Universal Robots PolyScope program: Cobot_soudure_28112023.urp

Program Cobot_soudure_28112023 (installation=Cobot_soudure_28112023 directory=/home/ur/ursim/ursim-5.11.0.108249/programs/TRAVAIL 27112023 createdIn=5.9.4.1031232 lastSavedIn=5.11.0.108249 robotSerialNumber=20195299999)
Calibrated DH parameters: a=[0, -0.6127, -0.57155, 0, 0, 0]; d=[0.1807, 0, 0, 0.17415, 0.11985, 0.11655]; alpha=[1.570796, 0, 0, 1.570796, -1.570796, 0]; deltaTheta=[0, 0, 0, 0, 0, 0]
InitVariablesNode variables(variable(name=Test_Gaz, expression=False), variable(name=Test_Job, expression=False), variable(name=Test_Ordre_Mar, expression=False), variable(name=Valide_Gaz, expression=False), variable(name=fin_soud, expression=1), variable(name=secu_d, expression=0), variable(name=secu_g, expression=0), variable(name=timer_ret_gaz, expression=0))
BeforeStart
  Folder fonctions
    Folder Init [hidden by the author, left out]
    Folder Diverses [hidden by the author, left out]
    Folder Demande [hidden by the author, left out]
    Folder Configuration [hidden by the author, left out]
    Folder Execution [hidden by the author, left out]
    Folder Pas_A_Pas [hidden by the author, left out]
    Folder PopUps [hidden by the author, left out]
    Folder Mouvements soudures [hidden by the author, left out]
    Folder General [hidden by the author, left out]
Robot Program (runOnlyOnce=true)
  SuppressedNode
    Script file /home/ur/ursim/ursim-5.11.0.108249/programs/SCRIPT/Scripts_soudure/general.script
      | while (True):
      |   # 68 "Programme de robot"
      |   global safe_mode=0
      | 
      |   set_configurable_digital_out(0, False)
      |   set_configurable_digital_out(1, False)
      | 
      |   while (get_configurable_digital_in(4) ==   True    or  get_configurable_digital_in(5) ==   True  ):
      | 
      |     sync()
      |     # 94 "'clingottement pour signifier qu'il y  un defaut sur un des carters '"
      |     set_standard_digital_out(4, False)
      |     set_configurable_digital_out(6, False)
      |     sleep(0.5)
      |     set_standard_digital_out(4, True)
      |     set_configurable_digital_out(6, True)
      |     sleep(0.5)
      |     sync()
      |   end
      | 
      |   set_configurable_digital_out(6, False)
      |   set_standard_digital_out(4, False)
      |   sleep(2.0)
      |   #movel(pose_add(get_target_tcp_pose(), pose_sub(PointPassage_12_to_p, PointPassage_12_from_p)), a=0.01, v=2.0E-4)
      |   global angle_base= get_actual_joint_positions ()
      |   if (angle_base[0]  <= 0.7):
      |     if (angle_base[0] >= 1.6):
      |       # 116 "Départ"        A CHANGER PAR UNE POSTION ENREGISTREE
      |       movej(pose_depart, a=accelerationHorsSoudure, v=vitesseHorsSoudure)
      |     else:
      |       if (angle_base[0]>1.6):
      |         movej(Point_init_D, a=accelerationHorsSoudure, v=vitesseHorsSoudure)
      |         movej(Point_avt_initD, a=accelerationHorsSoudure, v=vitesseHorsSoudure)
      |       else:
      |         if (angle_base[0]<0.7):
      |           movej(Point_init_G, a=accelerationHorsSoudure, v=vitesseHorsSoudure)
      |         end
      |       end
      |     end
      |   else:
      |     # 124 "SinonSi angle_base[0]>1.6"
      |     if (angle_base[0]>1.6):
      | 
      |       movej(Point_init_D, a=accelerationHorsSoudure, v=vitesseHorsSoudure)
      |       movej(Point_avt_initD, a=accelerationHorsSoudure, v=vitesseHorsSoudure)
      |     else:
      |       if (angle_base[0]<0.7):
      |         movej(Point_init_G, a=accelerationHorsSoudure, v=vitesseHorsSoudure)
      |       end
      |     end
      |   end
      |   # 131 "Départ"             A CHANGER PAR UNE POSTION ENREGISTREE
      |   movej(pose_depart, a=accelerationHorsSoudure, v=vitesseHorsSoudure)
      |   global angle_base= get_actual_joint_positions ()
      |   # 'mode config'
      |   if (get_configurable_digital_in(7)  ==   False    and  get_standard_digital_in(7)  ==   False  ):
      |     if ((config_g  ==  1)   and   (config_d  ==  1)):
      |       pop_up_config_g_et_d()
      |     else:
      |       if ((config_g  == 1)):
      |         pop_up_config_g()
      |       else:
      |         if (config_d  ==  1):
      |           pop_up_config_d()
      |         else:
      |           if ((config_g  ==  0)  and  (config_d  ==  0)):
      |             pop_up_config()
      |           end
      |         end
      |       end
      |     end
      |     global boucle=1
      |     while ((get_configurable_digital_in(7)  ==   False  )  and  (boucle  ==  1)   and  (get_standard_digital_in(7) ==   False  )):
      |       thread Thread_while_145():
      |         while (True):
      |           set_standard_digital_out(5, True)
      |           set_standard_digital_out(6, False)
      |           sleep(0.5)
      |           set_standard_digital_out(5, False)
      |           set_standard_digital_out(6, True)
      |           sleep(0.5)
      |           sync()
      |         end
      |       end
      |       if (get_standard_digital_in(3) ==   False    and  get_standard_digital_in(2) ==   False    and  get_configurable_digital_in(add_bp_ConfigReglage)  ==    False    and  get_standard_digital_in(add_bp_ConfigReglage) ==   False  ):
      |         global thread_handler_145=run Thread_while_145()
      |         while (get_standard_digital_in(3) ==   False    and  get_standard_digital_in(2) ==   False    and  get_configurable_digital_in(add_bp_ConfigReglage)  ==    False    and  get_standard_digital_in(add_bp_ConfigReglage) ==   False  ):
      |           sync()
      |         end
      |         kill thread_handler_145
      |       end
      |       if (get_standard_digital_in(2)  ==   True  ):
      |         set_standard_digital_out(5, True)
      |         set_standard_digital_out(6, False)
      |         movej(Point_init_G, a=accelerationHorsSoudure, v=vitesseHorsSoudure, r=0.006)
      |         movej(Point_Attente_G, a=accelerationHorsSoudure, v=vitesseHorsSoudure, r=0.006)
      |         movej(Point_config_g, a=accelerationHorsSoudure, v=vitesseHorsSoudure)
      |         global led_cobot=1
      |         fun_config_g()
      |         global led_cobot=0
      |         fun_valid_config_g()
      |         movej(Point_Attente_G, a=accelerationHorsSoudure, v=vitesseHorsSoudure, r=0.006)
      |         movej(Point_init_G, a=accelerationHorsSoudure, v=vitesseHorsSoudure, r=0.006)
      |         # 170 "Départ"         A CHANGER PAR UNE POSTION ENREGISTREE
      |         movej(pose_depart, a=accelerationHorsSoudure, v=vitesseHorsSoudure)
      |       end
      | 
      |       if (get_standard_digital_in(3)  ==   True  ):
      |         set_standard_digital_out(6, True)
      |         set_standard_digital_out(5, False)
      |         movej(Point_avt_initD, a=accelerationHorsSoudure, v=vitesseHorsSoudure, r=0.006)
      |         movej(Point_init_D, a=accelerationHorsSoudure, v=vitesseHorsSoudure)
      |         movej(Point_Attente_D, a=accelerationHorsSoudure, v=vitesseHorsSoudure, r=0.006)
      |         movej(Point_config_d, a=accelerationHorsSoudure, v=vitesseHorsSoudure)
      |         global led_cobot=1
      |         fun_config_d()
      |         global led_cobot=0
      |         fun_valid_config_d()
      |         movej(Point_Attente_D, a=accelerationHorsSoudure, v=vitesseHorsSoudure, r=0.006)
      |         movej(Point_init_D, a=accelerationHorsSoudure, v=vitesseHorsSoudure, r=0.006)
      |         movej(Point_avt_initD, a=accelerationHorsSoudure, v=vitesseHorsSoudure, r=0.006)
      |         # 190 "Départ"         A CHANGER PAR UNE POSTION ENREGISTREE
      |         movej(pose_depart, a=accelerationHorsSoudure, v=vitesseHorsSoudure)
      |       end
      |     end
      |   end
      |   # '"Reglage"'
      | 
      |   if (get_configurable_digital_in(add_bp_ConfigReglage)  ==   False    and  get_standard_digital_in(add_bp_ConfigReglage)  ==   True  ):
      |     if ((config_g  ==  1)   and   (config_d  ==  1)):
      |       pop_up_reg_gd()
      |       global boucle=1
      |     else:
      |       if (config_g  ==  1):
      |         pop_up_reg_gd()
      |         global boucle=1
      |       else:
      |         if (config_d  ==  1):
      |           pop_up_reg_d()
      |           global boucle=1
      |         else:
      |           close_popup()
      |           while (get_standard_digital_in(add_bp_ConfigReglage)  ==   True  ):
      |             popup("Aucune configuration n'est actuellement detectée.", "Erreur", False, True, blocking=True)
      |           end
      |         end
      |       end
      |     end
      |     global boucle=1
      |     while ((get_configurable_digital_in(add_bp_ConfigReglage)  ==   False  )  and  (boucle  ==  1)   and  (get_standard_digital_in(add_bp_ConfigReglage) ==   True  )):
      |       thread Thread_while_208():
      |         while (True):
      |           if (config_g  ==  1):
      |             set_standard_digital_out(5, True)
      |           end
      |           if (config_d  ==  1):
      |             set_standard_digital_out(6, True)
      |           end
      |           sleep(0.5)
      |           set_standard_digital_out(5, False)
      |           set_standard_digital_out(6, False)
      |           sleep(0.5)
      |         end
      |       end
      |       if (get_standard_digital_in(3) ==   False    and  get_standard_digital_in(2) ==   False    and  get_configurable_digital_in(7)  ==    False    and  get_standard_digital_in(7)  ==   True  ):
      |         global thread_handler_208=run Thread_while_208()
      |         while (get_standard_digital_in(3) ==   False    and  get_standard_digital_in(2) ==   False    and  get_configurable_digital_in(7)  ==    False    and  get_standard_digital_in(7)  ==   True  ):
      |           sync()
      |         end
      |         kill thread_handler_208
      |       end
      |       if (get_standard_digital_in(2)  ==   True  ):
      |         global safe_mode=1
      |         set_standard_digital_out(5, True)
      |         set_standard_digital_out(6, False)
      |         movej(Point_init_G, a=accelerationHorsSoudure, v=vitesseHorsSoudure, r=0.006)
      |         movej(Point_Attente_G, a=accelerationHorsSoudure, v=vitesseHorsSoudure, r=0.006)
      |         movej(pose_inter_g, a=accelerationHorsSoudure, v=vitesseHorsSoudure)
      |         global led_cobot=1
      |         fun_Pas_A_Pas_g()
      |         global led_cobot=0
      |         global safe_mode=0
      |         global boucle=0
      |       end
      |       if (get_standard_digital_in(3)  ==   True  ):
      |         global safe_mode=1
      |         set_standard_digital_out(6, True)
      |         set_standard_digital_out(5, False)
      |         movej(Point_avt_initD, a=accelerationHorsSoudure, v=vitesseHorsSoudure, r=0.006)
      |         movej(Point_init_D, a=accelerationHorsSoudure, v=vitesseHorsSoudure, r=0.006)
      |         movej(pose_inter_d, a=accelerationHorsSoudure, v=vitesseHorsSoudure)
      |         global led_cobot=1
      |         fun_Pas_A_Pas_d()
      |         global led_cobot=0
      |         global safe_mode=0
      |         global boucle=0
      |       end
      |     end
      |   end
      |   # 'mode execution'
      |   if (get_configurable_digital_in(add_bp_ConfigReglage)  ==   True  ):
      |     if ((config_g  ==  1)   and   (config_d  ==  1)):
      |       pop_up_exe()
      |       global boucle=1
      |     else:
      |       if (config_g  ==  1):
      |         pop_up_exe_g()
      |         global boucle=1
      |       else:
      |         if (config_d  ==  1):
      |           pop_up_exe_d()
      |           global boucle=1
      |         else:
      |           close_popup()
      |           while (get_configurable_digital_in(add_bp_ConfigReglage)  ==   True  ):
      |             popup("Aucune programmation n'est actuellement detectée, veillez à programmer une pièce avant de vouloir l'éxécuter.", "Erreur", False, True, blocking=True)
      |           end
      |         end
      |       end
      |     end
      |     while (( get_configurable_digital_in(add_bp_ConfigReglage)  ==   True  )   and  (boucle  ==  1)):
      |       thread Thread_while_259():
      |         while (True):
      |           if (config_g  ==  1):
      |             set_standard_digital_out(5, True)
      |           end
      |           if (config_d  ==  1):
      |             set_standard_digital_out(6, True)
      |           end
      |           sleep(0.5)
      |           set_standard_digital_out(5, False)
      |           set_standard_digital_out(6, False)
      |           sleep(0.5)
      |         end
      |       end
      |       if (get_standard_digital_in(3) ==   False    and  get_standard_digital_in(2) ==   False    and  get_configurable_digital_in(add_bp_ConfigReglage) ==   True  ):
      |         global thread_handler_259=run Thread_while_259()
      |         while (get_standard_digital_in(3) ==   False    and  get_standard_digital_in(2) ==   False    and  get_configurable_digital_in(add_bp_ConfigReglage) ==   True  ):
      |           sync()
      |         end
      |         kill thread_handler_259
      |       end
      |       if ((get_standard_digital_in(2)  ==   True  )  and  (config_g  ==   True  )):
      |         global boucle_g=1
      |         while (boucle_g  ==  1):
      |           set_configurable_digital_out(0, True)
      |           set_standard_digital_out(5, True)
      |           set_standard_digital_out(6, False)
      |           sleep(0.25)
      |           set_standard_digital_out(5, False)
      |           sleep(0.25)
      |           if (get_configurable_digital_in(4)  ==    False  ):
      |             set_standard_digital_out(5, True)
      |             if (get_configurable_digital_in(4)  ==    False  ):
      |               close_popup()
      |               while (get_configurable_digital_in(4) == False):
      |                 sync()
      |               end
      |             end
      |           end
      |           if (get_configurable_digital_in(4)  ==    True  ):
      |             global secu_g=1
      |             set_standard_digital_out(5, True)
      |             movej(Point_init_G, a=accelerationHorsSoudure, v=vitesseHorsSoudure, r=0.006)
      |             fun_execution_g()
      |             movej(Point_Attente_G, a=accelerationHorsSoudure, v=vitesseHorsSoudure, r=0.006)
      |             movej(Point_init_G, a=accelerationHorsSoudure, v=vitesseHorsSoudure, r=0.006)
      |             # 294 "Départ"         A CHANGER PAR UNE POSTION ENREGISTREE
      |             movej(pose_depart, a=accelerationHorsSoudure, v=vitesseHorsSoudure)
      |             set_configurable_digital_out(0, False)
      |             global secu_g=0
      |             global boucle_g=0
      |           end
      |         end
      |         global boucle=0
      |       else:
      |         if ((get_standard_digital_in(2)  ==   True  )  and  (config_g  ==   False  )):
      |           close_popup()
      |           popup("Aucune programmation n'est actuellement detectée sur la table gauche, veillez à programmer une pièce avant de vouloir l'éxécuter.", "Erreur", False, True, blocking=True)
      |           global boucle=0
      |         end
      |       end
      |       if ((get_standard_digital_in(3)  ==   True  )  and  (config_d  ==   True  )):
      |         global boucle_d=1
      |         pop_up_deb_exe_d()
      |         while (boucle_d  ==  1):
      |           set_configurable_digital_out(1, True)
      |           set_standard_digital_out(5, False)
      |           set_standard_digital_out(6, True)
      |           sleep(0.25)
      |           set_standard_digital_out(6, False)
      |           sleep(0.25)
      |           if (get_configurable_digital_in(5)  ==    False  ):
      |             set_standard_digital_out(6, True)
      |             sleep(6.0)
      |             if (get_configurable_digital_in(5)  ==    False  ):
      |               close_popup()
      |               while (get_configurable_digital_in(5) == False):
      |                 sync()
      |               end
      |             end
      |           end
      |           if (get_configurable_digital_in(5)  ==    True  ):
      |             global secu_d=1
      |             set_standard_digital_out(6, True)
      |             movej(Point_avt_initD, a=accelerationHorsSoudure, v=vitesseHorsSoudure)
      |             fun_execution_d()
      |             set_configurable_digital_out(1, False)
      |             global secu_d=0
      |             global boucle_d=0
      |           end
      |         end
      |         global boucle=0
      |       else:
      |         if ((get_standard_digital_in(3)  ==   True  )  and  (config_d  ==   False  )):
      |           close_popup()
      |           popup("Aucune programmation n'est actuellement detectée sur la table droite, veillez à programmer une pièce avant de vouloir l'éxécuter.", "Erreur", False, True, blocking=True)
      |           global boucle=0
      |         end
      |       end
      |     end
      |   end
      | end
      | end
  Script: General()
SubProgram Recopie_Table_Droite (keepSynchronizedWithDisk=false)
  SuppressedNode
    URCap Path (Robotiq_Copilot, Robotiq Inc.) dataModel(NodeInitializedKey=true, urcapVersion=1.14.3, pathOptionsTypeKey=TOOL_ON_ROBOT, HackTriggeringContributionIsDefinedMethodKey=true, version=1.14.3.2973, trajectoryPath={}); state(isChildrenLocked=true)
      URCap BeforeStart Node (Robotiq_Copilot, Robotiq Inc.)
        'Insert nodes below.'
  Popup Message (haltProgram=false message=Recopie sur la table de droite  inputType=Text)
SubProgram Recopie_Table_Gauche (keepSynchronizedWithDisk=false)
  SuppressedNode
    URCap Path (Robotiq_Copilot, Robotiq Inc.) dataModel(NodeInitializedKey=true, urcapVersion=1.14.3, pathOptionsTypeKey=TOOL_ON_ROBOT, HackTriggeringContributionIsDefinedMethodKey=true, version=1.14.3.2973, trajectoryPath={}); state(isChildrenLocked=true)
      URCap BeforeStart Node (Robotiq_Copilot, Robotiq Inc.)
        'Insert nodes below.'
  Popup Message (haltProgram=false message=Recopie sur la table de gauche inputType=Text)
Thread Thread_1 (runOnlyOnce=false)
  Folder Test_Ordre_Marche [hidden by the author, left out]
  Script: sync()
Thread Thread_2 (runOnlyOnce=false)
  Folder mode_soudure [hidden by the author, left out]
  Script: sync()
Thread Thread_3 (runOnlyOnce=false)
  Folder led_cobot_2 [hidden by the author, left out]
  Script: sync()
Thread Thread_4 (runOnlyOnce=false)
  Folder led_cobot [hidden by the author, left out]
  Script: sync()
Thread Thread_5 (runOnlyOnce=false)
  Folder Test_Arc_On [hidden by the author, left out]
  Script: sync()
Thread Thread_6 (runOnlyOnce=false)
  Folder Test_Job [hidden by the author, left out]
  Script: sync()
Thread Thread_7 (runOnlyOnce=false)
  Folder secu [hidden by the author, left out]
  Script: sync()
Thread Thread_8 (runOnlyOnce=false)
  Folder bloq_soud_arret [hidden by the author, left out]
  SuppressedNode
    Folder freedrive_droit
      If led_cobot ≟  True
        If tool_in[1] ≟ True
          Script: teach_mode()
        Else 
          Script: end_teach_mode()
  Script: sync()
SuppressedNode
  Thread Thread_9 (runOnlyOnce=false)
    Folder reglage
      If reglage_d ≠0
        Script file /programs/Programmes/cobot_v2/sript/Part_reglage/REGLAGE_D.script
          |     ##############################################################################
          | 
          | ########################soudure point#########################################
          | 
          |     ##############################################################################
          | 
          |         if reglage_d == 1:                                    #remplissage tableau
          |             teach_mode()
          |             fun_popup_soud(1, 1, i)
          |             fun_front_up(adresse_bp_cobot)
          |             tab_point_app_d[i] =  get_actual_tcp_pose()     #Enregistrer position dans tableau d'approche des soudue points quand appui bouton
          |             close_popup()
          | 
          |             fun_popup_soud(2, 1, i)
          |             fun_front_up(adresse_bp_cobot)
          |             tab_point_deb_d[i] =  get_actual_tcp_pose()     #Enregistrer position debut quand appui bouton bp_cobot
          |             close_popup()
          | 
          |             tab_point_ret_d[i] = tab_point_app_d[i]         #point de retrait est le meme que le point d approche
          |             end_teach_mode()
          |             global reconfig = 1
          |             global reglage_d = 0
          | 
          |             sync()
          | 
          |         ##############################################################################
          | 
          |     ##############################################################################
          | 
          | ########################soudure lineaire######################################
          | 
          |     ##############################################################################
          | 
          |         elif reglage_d == 2:                		            #remplissage tableau
          |             teach_mode()
          |             fun_popup_soud(1, 2, j)
          |             fun_front_up(adresse_bp_cobot)
          |             tab_lin_app_d[j] =  get_actual_tcp_pose()     	#Enregistrer position dans tableau d approche des soudures lineaire quand appui Bp_cobot
          |             close_popup()
          | 
          |             fun_popup_soud(2, 2, j)
          |             fun_front_up(adresse_bp_cobot)
          |             tab_lin_deb_d[j] =  get_actual_tcp_pose()     	#Enregistrer position dans tableau debut quand appui Bp_cobot
          |             close_popup()
          | 
          |             fun_popup_soud(6, 2, j)
          |             fun_front_up(adresse_bp_cobot)
          |             tab_lin_fin_d[j] =  get_actual_tcp_pose()     	#Enregistrer position dans un tableau fin quand appui Bp_cobot
          |             close_popup()
          | 
          |             vit_lin_d[j] = fun_demande_vit(2)
          | 
          |             fun_popup_soud(7, 2, j)
          |             fun_front_up(adresse_bp_cobot)
          |             tab_lin_ret_d[j] =  get_actual_tcp_pose()     	#Enregistrer position dans tableau retrait quand appui Bp_cobot
          |             close_popup()
          |             end_teach_mode()
          |             global reglage_d = 0
          | 
          |             sync()
          | 
          |         ##############################################################################
          | 
          |     ##############################################################################
          | 
          | #########################soudure arc de cercle##################################
          | 
          |     #################################################################################
          | 
          |         elif reglage_d == 3:                                  #remplissage tableau
          |             teach_mode()
          |             fun_popup_soud(1, 3, k)
          |             fun_front_up(adresse_bp_cobot)
          |             tab_arc_app_d[k] =  get_actual_tcp_pose() 	    #Enregistrer position dans tableau d approche des soudures arc de cercle quand appui
          |             close_popup()
          | 
          |             fun_popup_soud(2, 3, k)
          |             fun_front_up(adresse_bp_cobot)
          |             tab_arc_deb_d[k] =  get_actual_tcp_pose() 	    #Enregistrer position dans tableau debut quand appui Bp_d
          |             close_popup()
          | 
          |             fun_popup_soud(4, 3, k)
          |             fun_front_up(adresse_bp_cobot)
          |             tab_arc_mil_d[k] =  get_actual_tcp_pose() 	    #Enregistrer position dans tableau milieu quand appui Bp_cobot
          |             close_popup()
          | 
          |             fun_popup_soud(6, 3, k)
          |             fun_front_up(adresse_bp_cobot)
          |             tab_arc_fin_d[k] =  get_actual_tcp_pose() 	    #Enregistrer position dans un tableau fin quand appui Bp_cobot
          |             close_popup()
          | 
          |             vit_arc_d[k] = fun_demande_vit(3)               #demande de vitesse des soudures lineaire
          | 
          |             fun_popup_soud(7, 3, k)
          |             fun_front_up(adresse_bp_cobot)
          |             tab_arc_ret_d[k] =  get_actual_tcp_pose() 	    #Enregistrer position dans tableau retrait quand appui Bp_cobot
          |             close_popup()
          |             end_teach_mode()
          |             global reglage_d = 0
          | 
          |             sync()
          | 
          |         ##############################################################################
          | 
          |     ##############################################################################
          | 
          | ############################soudure cercle####################################
          | 
          |     #################################################################################
          | 
          |         elif reglage_d == 4:                                  #remplissage tableau
          |             teach_mode()
          |             fun_popup_soud(1, 4, l)
          |             fun_front_up(adresse_bp_cobot)
          |             tab_cer_app_d[l] =  get_actual_tcp_pose()     	#Enregistrer position dans tableau d approche des soudures arc de cercle quand appui Bp_cobot
          |             close_popup()
          | 
          |             fun_popup_soud(2, 4, l)
          |             fun_front_up(adresse_bp_cobot)
          |             tab_cer_deb_d[l] =  get_actual_tcp_pose()     	#Enregistrer position dans tableau debut quand appui Bp_cobot
          |             close_popup()
          | 
          |             fun_popup_soud(3, 4, l)
          |             fun_front_up(adresse_bp_cobot)
          |             tab_cer_quart_d[l] =  get_actual_tcp_pose()   	#Enregistrer position dans tableau d'approche des soudures arc de cercle quand appui Bp_d
          |             close_popup()
          | 
          |             fun_popup_soud(4, 4, l)
          |             fun_front_up(adresse_bp_cobot)
          |             tab_cer_mil_d[l] =  get_actual_tcp_pose()     	#Enregistrer position dans tableau milieu quand appui Bp_cobot
          |             close_popup()
          | 
          |             fun_popup_soud(5, 4, l)
          |             fun_front_up(adresse_bp_cobot)
          |             tab_cer_tro_d[l] =  get_actual_tcp_pose()     	#Enregistrer position dans tableau milieu quand appui Bp_cobot
          |             close_popup()
          | 
          |             fun_popup_soud(6, 4, l)
          |             fun_front_up(adresse_bp_cobot)
          |             tab_cer_fin_d[l] =  get_actual_tcp_pose()     	#Enregistrer position dans un tableau fin quand appui Bp_cobot
          |             close_popup()
          | 
          |             vit_cer_d[l] = fun_demande_vit(4)
          | 
          |             fun_popup_soud(7, 4, l)
          |             fun_front_up(adresse_bp_cobot)
          |             tab_cer_ret_d[l] =  get_actual_tcp_pose()    	#position de retrait est la meme que position d approche
          |             close_popup()
          |             end_teach_mode()
          |             global reglage_d = 0
          |             sync()
          | 
          |         end
          | 
          |     ##############################################################################
          | 
          | ############################################################
        Script: sync()
      If reglage_g ≠0
        Script file /programs/usbdisk_0/COBOT/finish/reg/REGLAGE_G.script
          |     ##############################################################################
          | 
          | ########################soudure point#########################################
          | 
          |     ##############################################################################
          | 
          |         if reglage_g == 1:                                    #remplissage tableau
          |             teach_mode()
          |             fun_popup_soud(1, 1, i)
          |             fun_front_up(adresse_bp_cobot)
          |             tab_point_app_g[i] =  get_actual_tcp_pose()     #Enregistrer position dans tableau d'approche des soudue points quand appui bouton
          |             close_popup()
          | 
          |             fun_popup_soud(2, 1, i)
          |             fun_front_up(adresse_bp_cobot)
          |             tab_point_deb_g[i] =  get_actual_tcp_pose()     #Enregistrer position debut quand appui bouton bp_cobot
          |             close_popup()
          | 
          |             tab_point_ret_g[i] = tab_point_app_g[i]         #point de retrait est le meme que le point d approche
          |             end_teach_mode()
          |             global reconfig = 1
          |             global reglage_g = 0
          | 
          |             sync()
          | 
          |         ##############################################################################
          | 
          |     ##############################################################################
          | 
          | ########################soudure lineaire######################################
          | 
          |     ##############################################################################
          | 
          |         elif reglage_g == 2:                		            #remplissage tableau
          |             teach_mode()
          |             fun_popup_soud(1, 2, j)
          |             fun_front_up(adresse_bp_cobot)
          |             tab_lin_app_g[j] =  get_actual_tcp_pose()     	#Enregistrer position dans tableau d approche des soudures lineaire quand appui Bp_cobot
          |             close_popup()
          | 
          |             fun_popup_soud(2, 2, j)
          |             fun_front_up(adresse_bp_cobot)
          |             tab_lin_deb_g[j] =  get_actual_tcp_pose()     	#Enregistrer position dans tableau debut quand appui Bp_cobot
          |             close_popup()
          | 
          |             fun_popup_soud(6, 2, j)
          |             fun_front_up(adresse_bp_cobot)
          |             tab_lin_fin_g[j] =  get_actual_tcp_pose()     	#Enregistrer position dans un tableau fin quand appui Bp_cobot
          |             close_popup()
          | 
          |             vit_lin_g[j] = fun_demande_vit(2)
          | 
          |             fun_popup_soud(7, 2, j)
          |             fun_front_up(adresse_bp_cobot)
          |             tab_lin_ret_g[j] =  get_actual_tcp_pose()     	#Enregistrer position dans tableau retrait quand appui Bp_cobot
          |             close_popup()
          |             end_teach_mode()
          |             global reglage_g = 0
          | 
          |             sync()
          | 
          |         ##############################################################################
          | 
          |     ##############################################################################
          | 
          | #########################soudure arc de cercle##################################
          | 
          |     #################################################################################
          | 
          |         elif reglage_g == 3:                                  #remplissage tableau
          |             teach_mode()
          |             fun_popup_soud(1, 3, k)
          |             fun_front_up(adresse_bp_cobot)
          |             tab_arc_app_g[k] =  get_actual_tcp_pose() 	    #Enregistrer position dans tableau d approche des soudures arc de cercle quand appui
          |             close_popup()
          | 
          |             fun_popup_soud(2, 3, k)
          |             fun_front_up(adresse_bp_cobot)
          |             tab_arc_deb_g[k] =  get_actual_tcp_pose() 	    #Enregistrer position dans tableau debut quand appui BP_cobot
          |             close_popup()
          | 
          |             fun_popup_soud(4, 3, k)
          |             fun_front_up(adresse_bp_cobot)
          |             tab_arc_mil_g[k] =  get_actual_tcp_pose() 	    #Enregistrer position dans tableau milieu quand appui Bp_cobot
          |             close_popup()
          | 
          |             fun_popup_soud(6, 3, k)
          |             fun_front_up(adresse_bp_cobot)
          |             tab_arc_fin_g[k] =  get_actual_tcp_pose() 	    #Enregistrer position dans un tableau fin quand appui Bp_cobot
          |             close_popup()
          | 
          |             vit_arc_g[k] = fun_demande_vit(3)               #demande de vitesse des soudures lineaire
          | 
          |             fun_popup_soud(7, 3, k)
          |             fun_front_up(adresse_bp_cobot)
          |             tab_arc_ret_g[k] =  get_actual_tcp_pose() 	    #Enregistrer position dans tableau retrait quand appui Bp_cobot
          |             close_popup()
          |             end_teach_mode()
          |             global reglage_g = 0
          | 
          |             sync()
          | 
          |         ##############################################################################
          | 
          |     ##############################################################################
          | 
          | ############################soudure cercle####################################
          | 
          |     #################################################################################
          | 
          |         elif reglage_g == 4:                                  #remplissage tableau
          |             teach_mode()
          |             fun_popup_soud(1, 4, l)
          |             fun_front_up(adresse_bp_cobot)
          |             tab_cer_app_g[l] =  get_actual_tcp_pose()     	#Enregistrer position dans tableau d approche des soudures arc de cercle quand appui Bp_cobot
          |             close_popup()
          | 
          |             fun_popup_soud(2, 4, l)
          |             fun_front_up(adresse_bp_cobot)
          |             tab_cer_deb_g[l] =  get_actual_tcp_pose()     	#Enregistrer position dans tableau debut quand appui Bp_cobot
          |             close_popup()
          | 
          |             fun_popup_soud(3, 4, l)
          |             fun_front_up(adresse_bp_cobot)
          |             tab_cer_quart_g[l] =  get_actual_tcp_pose()   	#Enregistrer position dans tableau d'approche des soudures arc de cercle quand appui Bp_cobot
          |             close_popup()
          | 
          |             fun_popup_soud(4, 4, l)
          |             fun_front_up(adresse_bp_cobot)
          |             tab_cer_mil_g[l] =  get_actual_tcp_pose()     	#Enregistrer position dans tableau milieu quand appui Bp_cobot
          |             close_popup()
          | 
          |             fun_popup_soud(5, 4, l)
          |             fun_front_up(adresse_bp_cobot)
          |             tab_cer_tro_g[l] =  get_actual_tcp_pose()     	#Enregistrer position dans tableau milieu quand appui Bp_cobot
          |             close_popup()
          | 
          |             fun_popup_soud(6, 4, l)
          |             fun_front_up(adresse_bp_cobot)
          |             tab_cer_fin_g[l] =  get_actual_tcp_pose()     	#Enregistrer position dans un tableau fin quand appui Bp_cobot
          |             close_popup()
          | 
          |             vit_cer_g[l] = fun_demande_vit(4)
          | 
          |             fun_popup_soud(7, 4, l)
          |             fun_front_up(adresse_bp_cobot)
          |             tab_cer_ret_g[l] =  get_actual_tcp_pose()    	#position de retrait est la meme que position d approche
          |             close_popup()
          |             end_teach_mode()
          |             global reglage_g = 0
          |             sync()
          | 
          |         end
          | 
          |     ##############################################################################
          | 
          | ############################################################
        Script: sync()
      Script: sync()
    Script: sync()
Thread Thread_10 (runOnlyOnce=false)
  Folder reglage [hidden by the author, left out]
  Script: sync()
